// Subject under test
FUNCTION_BLOCK INTERNAL FB_XV03ValveSystem_Tests EXTENDS FB_TestSuite

// Create instance variables that will be accesible for all tests
VAR

END_VAR

// Call your test methods here
Test01_Disabled_AllOutputsAreAlwaysFalse();
Test02_Enabled_ExpectCorrectByteBitsSetToTrue();

METHOD PRIVATE Test01_Disabled_AllOutputsAreAlwaysFalse

(* Instanced variables are VERY useful for writing tests since tests are run in paralel (by default).
By instantiating local variables that are not placed on the same stack as method (values are retained between calls)
you make sure that the SUT is not changed by some other test. *)
VAR_INST
	emptyArray	: ARRAY[0..SIZEOF(ST_ValveCoils)] OF BYTE;
	fbValves	: FB_XV03_ValveSystem(0);
END_VAR

VAR_INST

END_VAR
// The name of the test, is the same as method name!
IF TcUnit.TEST_ORDERED('Test01_Disabled_AllOutputsAreAlwaysFalse') THEN
	fbValves.Enable := FALSE;
	
	AssertTrue(
		Condition := Tc2_System.MEMCMP(pBuf1 := ADR(emptyArray), pBuf2 := ADR(fbValves.Coils), n := SIZEOF(ST_ValveCoils))  = ZigaLibs_Core.E_MemCmpResults.IDENTICAL,
		Message := 'When disabled, output coils should all be set to 0.');
		
	fbValves.Valves[1].Coil_12.Active := TRUE;
	fbValves.Valves[5].Coil_14.Active := TRUE;
	fbValves.Valves[8].Coil_12.Active := TRUE;
	fbValves.Valves[12].Coil_12.Active := TRUE;
	
	AssertTrue(
		Condition := Tc2_System.MEMCMP(
			pBuf1 := ADR(emptyArray), 
			pBuf2 := ADR(fbValves.Coils), 
			n := SIZEOF(ST_ValveCoils)) = ZigaLibs_Core.E_MemCmpResults.IDENTICAL,
		Message := 'When disabled, output coils should all be set to 0.');

	TcUnit.TEST_FINISHED();	
END_IF
END_METHOD

METHOD PRIVATE Test02_Enabled_ExpectCorrectByteBitsSetToTrue

(* Instanced variables are VERY useful for writing tests since tests are run in paralel (by default).
By instantiating local variables that are not placed on the same stack as method (values are retained between calls)
you make sure that the SUT is not changed by some other test. *)
VAR_INST
		fbValveSystem_XV03	: FB_XV03_ValveSystem(0);
END_VAR

VAR
	iteration						: UINT;
	ptrUsint						: POINTER TO USINT;
	indexValueToAdd					: UINT;
	indexValueToSubstract			: UINT;
	expectedValue					: USINT;
	stringBuilder					: ZigaLibs_Core.FB_StringBuilder;
	addressToAdd					: DWORD;
END_VAR

VAR CONSTANT
	VALVES_PER_BYTE	: REAL := 4.0;
END_VAR
// The name of the test, is the same as method name!
IF TcUnit.TEST_ORDERED('Test02_Enabled_ExpectCorrectByteBitsSetToTrue') THEN
	fbValveSystem_XV03.Enable := TRUE;
	
	FOR iteration := 1 TO 24 BY 1 DO
		// Coil 1 of valve
		fbValveSystem_XV03.Valves[iteration].Coil_14.Active := TRUE;
		fbValveSystem_XV03();
		// add + 1 address when next byte should be looked at (4 valves with 2 coils per byte, 8 bits)
		addressToAdd := LREAL_TO_DWORD((Tc2_Math.FLOOR(TO_LREAL(iteration - 1)/VALVES_PER_BYTE)));
		ptrUsint := ADR(fbValveSystem_XV03.Coils) + addressToAdd;
		expectedValue := LREAL_TO_USINT(EXPT(2, iteration - 1 + indexValueToAdd - indexValueToSubstract));
		AssertTrue(
			Condition := ptrUsint^ = expectedValue,
			Message := stringBuilder.Reset()
				.AddString('Valve ')
				.AddWithDblQuotationMarks(TO_STRING(iteration))
				.AddString(', coil 14 was not opened.')
				.Create());
		
		fbValveSystem_XV03.Valves[iteration].Coil_14.Active := FALSE;
		fbValveSystem_XV03();
		AssertTrue(
			Condition := ptrUsint^ = 0,
			Message := stringBuilder.Reset()
				.AddString('Valve ')
				.AddWithDblQuotationMarks(TO_STRING(iteration))
				.AddString(', coil 14 was not closed.')
				.Create());
		
		// Coil 2 of valve	
		fbValveSystem_XV03.Valves[iteration].Coil_12.Active := TRUE;
		fbValveSystem_XV03();
		// Every 4th valve proceeds to next byte (2 coils per valve, 2x4 = 8 bits = 1 byte, 48 coils total)
		addressToAdd := LREAL_TO_DWORD((Tc2_Math.FLOOR(TO_LREAL(iteration - 1)/VALVES_PER_BYTE)));
		ptrUsint := ADR(fbValveSystem_XV03.Coils) + addressToAdd;
		expectedValue := LREAL_TO_USINT(EXPT(2, iteration + indexValueToAdd - indexValueToSubstract));
		AssertTrue(ptrUsint^ = expectedValue,
			stringBuilder.Reset()
				.AddString('Valve ')
				.AddWithDblQuotationMarks(TO_STRING(iteration))
				.AddString(', coil 12 was not opened.')
				.Create());
				
		indexValueToAdd := indexValueToAdd + 1;
		
		fbValveSystem_XV03.Valves[iteration].Coil_12.Active := FALSE;
		fbValveSystem_XV03();
		AssertTrue(
			Condition := ptrUsint^ = 0,
			Message := stringBuilder.Reset()
				.AddString('Valve ')
				.AddWithDblQuotationMarks(TO_STRING(iteration))
				.AddString(', coil 12 was not closed.')
				.Create());
				
		// In order to have 1 single loop, every loop iteration we need to add 1 value, to increase the 2^n+1 result.
		// When the byte is finished, next iteration would start at 2^n, for example 2^5. But we need to reset back at 1st position.
		// For that reson the substract index will be taken into account in the power calculation and every 4th iteration, 
		// aka 1 byte, the power will be: 2^(iteration - 4*(byte number 0...3) + current coil index (0..1))		
		IF indexValueToAdd = TO_UINT(VALVES_PER_BYTE) THEN
			indexValueToAdd := 0;
			indexValueToSubstract := indexValueToSubstract + TO_UINT(VALVES_PER_BYTE);
		END_IF
	END_FOR
	
	TcUnit.TEST_FINISHED();
END_IF
END_METHOD

END_FUNCTION_BLOCK

(* stored: Version 1.1.0.1, ProductVersion 3.1.4024.16
   POU FB_XV03ValveSystem_Tests: Id {6e93b8ca-791a-0f0b-085c-81624b4b6d87}, SpecialFunc None
   Method Test01_Disabled_AllOutputsAreAlwaysFalse: Id {0eca35e2-db47-055a-20be-974be9dcb115}
   Method Test02_Enabled_ExpectCorrectByteBitsSetToTrue: Id {69a0d643-44bb-0985-2513-ae9bafacd361} *)
